TYPE ST_Selection :
STRUCT
	Select			: BOOL;
	Queued			: BOOL;
	Enabled	    	: BOOL;
	Interlock		: BOOL;
	Messages		: STRING[255];
	Description		: STRING[255];
END_STRUCT
END_TYPE

(* stored: Version 1.1.0.1, ProductVersion 3.1.4024.3
   DUT ST_Selection: Id {725e8aa0-451f-4ccf-913d-d3f43e6a160a} *)
